// TwinCAT 3 PLC project Untitled1
// ProgramVersion: 3.1.4024.0
// libraries:
//   Tc2_Standard, * (Beckhoff Automation GmbH)
//   Tc2_System, * (Beckhoff Automation GmbH)
//   Tc3_Module, * (Beckhoff Automation GmbH)
// project tree:
//   DUTs/ enm_state.TcDUT
//   GVLs/ IO.TcGVL
//   / PlcTask.TcTTO
//   POUs/ FB_StateMachine.TcPOU, MAIN.TcPOU
// real-time tasks:
//   TASK PlcTask: cycle T#10ms, priority 20, ADS port 350

CONFIGURATION Untitled1
    RESOURCE PLC ON TwinCAT3
        TASK PlcTask(INTERVAL := T#10ms, PRIORITY := 20);
        PROGRAM MAIN WITH PlcTask : MAIN;
    END_RESOURCE
END_CONFIGURATION

// ---- DUTs/enm_state.TcDUT
{attribute 'qualified_only'}
{attribute 'strict'}
TYPE enm_state :
(
	undifined := 0,
	Init,
	Automod,
	Manualmod
);
END_TYPE

// ---- GVLs/IO.TcGVL
{attribute 'qualified_only'}
VAR_GLOBAL
	bYellos_Mode 	AT %I*:BOOL;
	bBlue_Lamp 		AT %I* :BOOL;
	
	bGreenLight		AT %Q*:BOOL;
	bRedLight		AT %Q*:BOOL;
	
	iUltraschallSensor AT %I*:INT;
END_VAR

// ---- POUs/MAIN.TcPOU
PROGRAM MAIN
VAR
	fb_statemachine : FB_StateMachine;
END_VAR

fb_statemachine();

END_PROGRAM

// ---- POUs/FB_StateMachine.TcPOU
FUNCTION_BLOCK FB_StateMachine
VAR_INPUT
END_VAR
VAR_OUTPUT
END_VAR
VAR
	State:		enm_state := enm_state.Init;
	ton_timerAutoMode : Ton;
END_VAR

//noch ein Fehler man müsste noch warten bis der Taster wieder los gelassen ist.
CASE State OF
	enm_state.undifined:
	;
	enm_state.Init:
	IO.bGreenLight:= TRUE;
	IO.bRedLight:= TRUE;
	IF IO.bYellos_Mode THEN
		State := enm_state.Automod;

	END_IF
	;
	enm_state.Automod:
	ton_timerAutoMode(IN := TRUE, PT := T#2S);
	IF ton_timerAutoMode.Q = TRUE THEN
		IO.bRedLight := NOT IO.bRedLight;
		IO.bGreenLight:= NOT IO.bGreenLight;
		ton_timerAutoMode(IN := FALSE, PT := T#2S);
	END_IF
	
	IF IO.bYellos_Mode THEN
	State := enm_state.Init;
	END_IF
		
	;
	enm_state.Manualmod:
	;
END_CASE

END_FUNCTION_BLOCK
